{attribute 'qualified_only'}
VAR_GLOBAL
	AppConfig : AppConfig;
END_VAR

(* stored: Version 1.1.0.1, ProductVersion 3.1.4024.3
   GVL GlobalConfig: Id {fee94fa9-eed8-45f3-816b-23d1a714fcf3} *)
